// TIA Portal V19 export
TYPE "Positioning_MOL_Machine_DataIn"
// stored: Access Published
   STRUCT
      PB : "Ax_PB";
      LS_Minus : Bool;
      LS_Plus : Bool;
      M1_TherrmalProtection : Bool := FALSE;
      M2_TherrmalProtection : Bool := FALSE;   // Lasciare FALSE se non esiste
      M1M2_Feedback : Bool;
   END_STRUCT;
END_TYPE
